ABB RobotStudio station: step_smartcomponet_20200824-230510.rsstn

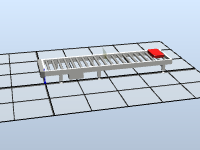
Station step_smartcomponet (saved by RobotStudio 6.8.8307.1040)
Controller IRB_120_3kg_0.58m_3
Layout (positions relative to the parent item):
  - IRB4600_60_205_C_01 [mechanism, from Robots\IRB4600_60_205_C_G_01.rslib] at (0, 0, 0) mm; joint values [0, 0, 0, 0, 0.5236, 0] (rad or m)
  - 950_4000_h2 [part, from Equipment\Conveyor 950 4000 h2.rslib]
  - CAJA [part, from Step_vacum_gripper\SOLCAJA.rslib] at (2900, 450, 412.42) mm
  - SmartComponent_1 [smart component]
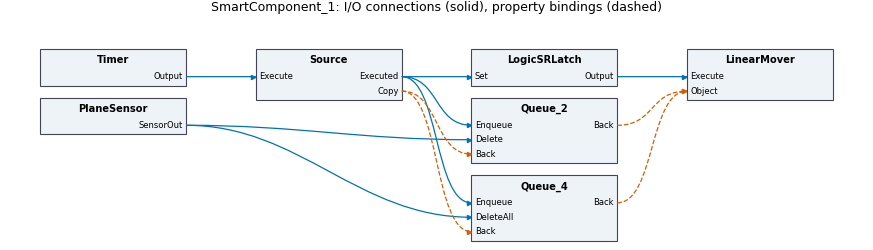
      connections:
        Timer.Output -> Source.Execute
        Source.Executed -> Queue_2.Enqueue
        LogicSRLatch.Output -> LinearMover.Execute
        PlaneSensor.SensorOut -> Queue_2.Delete
        Source.Executed -> Queue_4.Enqueue
        PlaneSensor.SensorOut -> Queue_4.DeleteAll
        Source.Executed -> LogicSRLatch.Set
        Source.Copy => Queue_2.Back
        Queue_2.Back => LinearMover.Object
        Source.Copy => Queue_4.Back
        Queue_4.Back => LinearMover.Object
    - Source [smart component, from Components\Source.rslib]
        properties: Source=CAJA; Copy=(none); Parent=(none); Position=[4.381792 2.252642 0]; Orientation=[0 0 0]; Transient=true; PhysicsBehavior=0
    - Timer [smart component, from Components\Timer.rslib]
        properties: StartTime=0; Interval=7; Repeat=true; CurrentTime=37.872
    - LinearMover [smart component, from Components\LinearMover.rslib]
        properties: Object=(none); Direction=[-1 0 0]; Speed=0.6; Reference=Global; ReferenceObject=(none)
    - PlaneSensor [smart component, from Components\PlaneSensor.rslib]
        properties: Origin=[2 0.1 0.45]; Axis1=[0 0.2 0.3]; Axis2=[0 0.5 0]; SensedPart=(none)
      - _sensorPart_ [part]
    - LogicSRLatch [smart component, from Components\LogicSRLatch.rslib]
    - Queue_4 [smart component, from Components\Queue.rslib]
        properties: Back=(none); Front=(none); Queue={c51ebb60-ab18-46a5-bcb4-c56f3e4f5d54};{e1eb26c3-23ea-4a3a-9c03-43a2b9c1cbfe};{a76681ba-1725-4bb8-860a-f3bac0ad59dc};{c111bf08-6e4c-46bf-8935-05d0526352b3};{5cc1aa04-befe-44fe-be44-3df6925351c4};{8fa9e6ac-08d3-4316-a911-1005c4ed7949};{52755cf1-1ecb-4d4d-b2dc-2ab09b9f28fa};{3f02d463-ed99-4175-a452-3989ed42dc9e};{0eb66b12-c7fd-4931-9696-25351aa88514};{105ec880-8e27-45cf-9e9a-fa92e7858842};{1ef477ec-cfaf-461a-aded-686da802c12c};{f9f47090-256a-4d62-9105-be76298c8d7a};{ac40bc69-9598-4231-96c8-b82ba84b5e74}; NumberOfObjects=5
